{attribute addProperty BoxType "KL8610-0007"}
{attribute addProperty Id "KL8601_1KL_B0A8062F00KL8601_2KL_B0A8062F00KL8601_3KL_B0A8062F00KL8601_4KL_B0A8062F00KL8601_5KL_B0A8062F00KL8601_6KL_B0A8062F00KL8601_7KL_B0A8062F00KL8601_8KL_B0A8062F00"}
{attribute addProperty CRC "1471797640"}
{attribute addProperty SizeInBites "0"}
{attribute addProperty SizeInBytes "0"}
TYPE KL_57B9D988 :
STRUCT
	{attribute addProperty Name "KL8601_1"}
	KL8601_1 : KL_B0A8062F;
	{attribute addProperty Name "KL8601_2"}
	KL8601_2 : KL_B0A8062F;
	{attribute addProperty Name "KL8601_3"}
	KL8601_3 : KL_B0A8062F;
	{attribute addProperty Name "KL8601_4"}
	KL8601_4 : KL_B0A8062F;
	{attribute addProperty Name "KL8601_5"}
	KL8601_5 : KL_B0A8062F;
	{attribute addProperty Name "KL8601_6"}
	KL8601_6 : KL_B0A8062F;
	{attribute addProperty Name "KL8601_7"}
	KL8601_7 : KL_B0A8062F;
	{attribute addProperty Name "KL8601_8"}
	KL8601_8 : KL_B0A8062F;
END_STRUCT
END_TYPE

(* stored: Version 1.2.0.0, ProductVersion 3.1.4024.9
   DUT KL_57B9D988: Id {53e0e3c5-01e9-443f-b4f8-c1e22012011b} *)
